// TIA Portal V19 export
FUNCTION "24 HOUR TIMER" : Void   // FC12, LAD
{ S7_Optimized_Access := 'TRUE' }
// stored: SetENOAutomatically false
   VAR_TEMP   // added for the SCL form of the ladder/FBD networks
      _w1 : Bool;
   END_VAR
BEGIN

REGION Network 1: 24 HOUR_TIMER
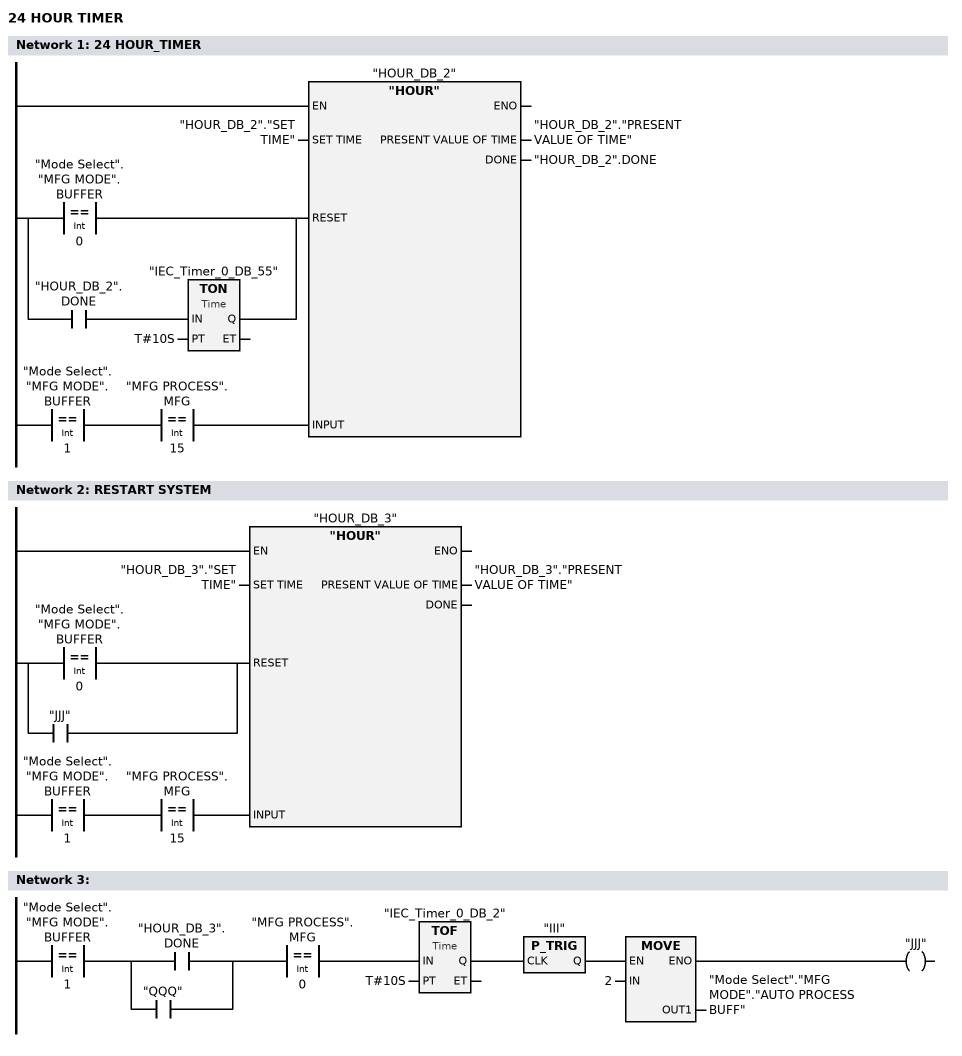
   RUNG wire#powerrail
      "HOUR_DB_2"(RESET := wire#w1, INPUT := wire#w2, "SET TIME" := "HOUR_DB_2"."SET TIME", "PRESENT VALUE OF TIME" => "HOUR_DB_2"."PRESENT VALUE OF TIME", DONE => "HOUR_DB_2".DONE)
   END_RUNG
   RUNG wire#powerrail
      { S7_Templates := "SrcType := Int" } EQ_Contact(in1 := "Mode Select"."MFG MODE".BUFFER, in2 := 0)
   END_RUNG wire#w1
   RUNG wire#powerrail
      Contact( "HOUR_DB_2".DONE )
      { S7_Templates := "time_type := Time" } "IEC_Timer_0_DB_55".TON(pt := T#10S, et =>)
   END_RUNG wire#w1
   RUNG wire#powerrail
      { S7_Templates := "SrcType := Int" } EQ_Contact(in1 := "Mode Select"."MFG MODE".BUFFER, in2 := 1)
      { S7_Templates := "SrcType := Int" } EQ_Contact(in1 := "MFG PROCESS".MFG, in2 := 15)
   END_RUNG wire#w2
   // the same network as SCL:
   "IEC_Timer_0_DB_55".TON(IN := "HOUR_DB_2".DONE, PT := T#10S);
   "HOUR_DB_2"("SET TIME" := "HOUR_DB_2"."SET TIME",   // "HOUR"
               RESET := ("Mode Select"."MFG MODE".BUFFER = 0) OR "IEC_Timer_0_DB_55".Q,
               INPUT := ("Mode Select"."MFG MODE".BUFFER = 1) AND ("MFG PROCESS".MFG = 15),
               "PRESENT VALUE OF TIME" => "HOUR_DB_2"."PRESENT VALUE OF TIME",
               DONE => "HOUR_DB_2".DONE);
END_REGION

REGION Network 2: RESTART SYSTEM
   RUNG wire#powerrail
      "HOUR_DB_3"(RESET := wire#w1, INPUT := wire#w2, "SET TIME" := "HOUR_DB_3"."SET TIME", "PRESENT VALUE OF TIME" => "HOUR_DB_3"."PRESENT VALUE OF TIME", DONE =>)
   END_RUNG
   RUNG wire#powerrail
      { S7_Templates := "SrcType := Int" } EQ_Contact(in1 := "Mode Select"."MFG MODE".BUFFER, in2 := 0)
   END_RUNG wire#w1
   RUNG wire#powerrail
      Contact( "JJJ" )
   END_RUNG wire#w1
   RUNG wire#powerrail
      { S7_Templates := "SrcType := Int" } EQ_Contact(in1 := "Mode Select"."MFG MODE".BUFFER, in2 := 1)
      { S7_Templates := "SrcType := Int" } EQ_Contact(in1 := "MFG PROCESS".MFG, in2 := 15)
   END_RUNG wire#w2
   // the same network as SCL:
   "HOUR_DB_3"("SET TIME" := "HOUR_DB_3"."SET TIME",   // "HOUR"
               RESET := ("Mode Select"."MFG MODE".BUFFER = 0) OR "JJJ",
               INPUT := ("Mode Select"."MFG MODE".BUFFER = 1) AND ("MFG PROCESS".MFG = 15),
               "PRESENT VALUE OF TIME" => "HOUR_DB_3"."PRESENT VALUE OF TIME");
END_REGION

REGION Network 3
   RUNG wire#powerrail
      { S7_Templates := "SrcType := Int" } EQ_Contact(in1 := "Mode Select"."MFG MODE".BUFFER, in2 := 1)
      wire#w1
      Contact( "HOUR_DB_3".DONE )
      wire#w2
      { S7_Templates := "SrcType := Int" } EQ_Contact(in1 := "MFG PROCESS".MFG, in2 := 0)
      { S7_Templates := "time_type := Time" } "IEC_Timer_0_DB_2".TOF(pt := T#10S, et =>)
      P_Trig( "III" )
      Move(in := 2, out1 => "Mode Select"."MFG MODE"."AUTO PROCESS BUFF")
      Coil( "JJJ" )
   END_RUNG
   RUNG wire#w1
      Contact( "QQQ" )
   END_RUNG wire#w2
   // the same network as SCL:
   "IEC_Timer_0_DB_2".TOF(IN := ("Mode Select"."MFG MODE".BUFFER = 1) AND ("HOUR_DB_3".DONE OR "QQQ") AND ("MFG PROCESS".MFG = 0),
                          PT := T#10S);
   #_w1 := "IEC_Timer_0_DB_2".Q AND NOT "III";   // rising edge
   "III" := "IEC_Timer_0_DB_2".Q;
   IF #_w1 THEN "Mode Select"."MFG MODE"."AUTO PROCESS BUFF" := 2; END_IF;
   "JJJ" := #_w1;
END_REGION
END_FUNCTION
